Fanuc KAREL source: ks00006.KL

-- PROVISIONAL review KL for V1013-1; original PC SHA256 1f687eece312ce454d41bb2c1e96b986e7e1833b65bffa9eb565cce2017fadd2
-- Incomplete behavior may be omitted. Consult companion uncertainty JSON. Do not deploy.
PROGRAM KS00006
%NOLOCKGROUP
VAR
  FLAG : BOOLEAN
  N : INTEGER
  STATUS : INTEGER
  PN : STRING[80]
  VN : STRING[80]
-- UNRESOLVED_DECL A type=001100
-- UNRESOLVED_DECL B type=001100
BEGIN
  -- UNRESOLVED_PC offsets 5-13; opcodes 3F,75
  -- UNRESOLVED_PC offsets 18-27; opcodes 3F,75
  -- UNRESOLVED_PC offsets 32-70; opcodes 27,22,22,2A,22,2A,22,22,AF
  -- UNRESOLVED_PC offsets 75-79; opcodes 7F
END KS00006
